FUNCTION_BLOCK FB_Dil_GetValveConfig
VAR_INPUT
	bExecute	: BOOL;	
END_VAR
VAR_OUTPUT
	bBusy		: BOOL;
	bError		: BOOL;
	nErrorId	: ERRORID;
	nValue		: USINT;
END_VAR
VAR
END_VAR
VAR_IN_OUT
	DilSendCmd 	: FB_Dil_SendCmd;
	pDilRef		: POINTER TO FB_HwRefDiluter;
END_VAR

IF pDilRef = 0 THEN
	bError := TRUE;
	RETURN;	
END_IF

IF bExecute THEN
	bBusy := TRUE;

	DilSendCmd(bExecute:= TRUE, bExpectReply:= TRUE, sSendData:= CONCAT(USINT_TO_STRING(pDilRef^.nChannel),'?21'));
	
	IF NOT DilSendCmd.bBusy THEN
		IF DilSendCmd.bError THEN
			bError := TRUE;
			nErrorId := DilSendCmd.nErrorId;
		ELSE
			nValue := F_ToASC(LEFT(DilSendCmd.sReceiveData,1)) AND 16#0F;
			pDilRef^.eValveType := nValue;
		END_IF
		DilSendCmd(bExecute:= FALSE);
		bBusy := FALSE;
	END_IF
ELSE
	DilSendCmd(bExecute:= FALSE);
	bBusy := FALSE;
	bError := FALSE;
	nErrorId := 0;
	nValue := 0;
END_IF

END_FUNCTION_BLOCK

(* stored: Version 1.1.0.1, ProductVersion 3.1.4022.10
   POU FB_Dil_GetValveConfig: Id {7313fd23-5c05-4730-88a4-de979afda87e}, SpecialFunc None *)
